# B&R Automation Studio project NAINV104C00R8L515F00 (part 29)

#### Act_Background_Sequence.st - Do Not Change!!!
```iecst
 (** 2019-05-04 **)
ACTION Act_Background_Sequence:

	IF eStatus1 <> Error THEN

		IF p_bOpsRun = FALSE THEN
			p_bSndIncompl	:= TRUE;
		END_IF

		IF tyMsgTypeRcv.bStopTransport = TRUE THEN
			IF tyStopTransport.tyData.eTransferState = HermesTransferStateNotStarted THEN
				p_bSndNotStart	:= TRUE;
			ELSIF tyStopTransport.tyData.eTransferState = HermesTransferStateIncomplete THEN
				p_bSndIncompl	:= TRUE;
			END_IF
		END_IF

		bBlkDS := p_bHermesSwitchtoRvrseTransport;
		//Sequence
		fbSequenceDS.bRstState		:= bRstState;
		fbSequenceDS.bRdySnd		:= p_bRdySnd;
		fbSequenceDS.bBlkDS			:= bBlkDS;
		fbSequenceDS.bSndCompl		:= p_bSndCompl;
		fbSequenceDS.bSndIncompl	:= p_bSndIncompl;
		fbSequenceDS.bSndNotStart	:= p_bSndNotStart;
		fbSequenceDS.bFeatureBoardForecast	:= bFeatureBoardForecast; //Feature BoardForecast
		fbSequenceDS.bOpsRun	        	:= p_bOpsRun; //Machine in AutoMode
		fbSequenceDS.bSendBFId              := bSendBFId; //Send B.F with forecast ID, then block Hermes.eState until Downstream reply a MachineReady(Id) or MachineReady()
		fbSequenceDS.bBFIdSent              := bBFIdSent;
		fbSequenceDS.bSendBFNoID			:= bSendBFNoID;
		fbSequenceDS(bEn := TRUE);
		bUSRdy			:= fbSequenceDS.bUSRdy;
		bDSRdy			:= fbSequenceDS.bDSRdy;
		bTransporting	:= fbSequenceDS.bTransporting;
		bStopTransport	:= fbSequenceDS.bStopTransport;

		bUSGdRdy	:= (tyBoardAvailableSnd.tyAvl.bFailedBoard = FALSE) OR ((tyBoardAvailableSnd.tyAvl.bFailedBoard = TRUE) AND (tyBoardAvailableSnd.tyData.eFailedBoard <> HermesFailedBoard));

		bDSGdRdy	:= (tyMachineReady.tyAvl.bFailedBoard = FALSE) OR ((tyMachineReady.tyAvl.bFailedBoard = TRUE) AND (tyMachineReady.tyData.eFailedBoard <> HermesFailedBoard));

		IF fbSequenceDS.eState >= HermesStateNotAvailableNotReady THEN
			bHandshakeDone	:= TRUE;
		ELSE
			bHandshakeDone	:= FALSE;
		END_IF

		IF EDGEPOS(fbSequenceDS.eState = HermesStateTransporting) THEN
			p_bSndCompl		:= FALSE;
			p_bSndIncompl	:= FALSE;
			p_bSndNotStart	:= FALSE;
		END_IF

		IF fbSequenceDS.eMsgTypeSnd = HermesMsgTypeServiceDescription THEN
			fHermesAddOneMsgSend(ADR(a_eMsgSend) , ADR(udiMsgSendBffr) , HermesMsgTypeServiceDescription);

			tyServiceDescriptionSnd.tyData.sMachineId								    	:= p_sMcId;
			tyServiceDescriptionSnd.tyData.iLaneId											:= p_tyParam.iLaneID;
			tyServiceDescriptionSnd.tyData.sInterfaceId										:= p_sInterfaceId;
			tyServiceDescriptionSnd.tyData.sVersion											:= p_sVersion;
			tyServiceDescriptionSnd.tyData.tySupportedFeatures.bFeatureCheckAliveResponse	:= (p_tyParam.bFeatureCheckAliveResponse) AND (p_tyParam.tRcvAlive <> T#0s) AND (p_tyParam.tSndAlive <> T#0s);
			tyServiceDescriptionSnd.tyData.tySupportedFeatures.bFeatureBoardForecast		:= p_tyParam.bFeatureBoardForecast;
			tyServiceDescriptionSnd.tyData.tySupportedFeatures.bFeatureQueryBoardInfo		:= FALSE;
			tyServiceDescriptionSnd.tyData.tySupportedFeatures.bFeatureSendBoardInfo		:= p_tyParam.bFeatureSendBoardInfo;
			tyServiceDescriptionSnd.tyData.tySupportedFeatures.bFeatureCommand				:= p_tyParam.bFeatureCommand;

			tyServiceDescriptionSnd.tyAvl.bMachineId										:= tyServiceDescriptionSnd.tyData.sMachineId <> '';
			tyServiceDescriptionSnd.tyAvl.bLaneId											:= tyServiceDescriptionSnd.tyData.iLaneId<>0;
			tyServiceDescriptionSnd.tyAvl.bInterfaceId										:= tyServiceDescriptionSnd.tyData.sInterfaceId <> '';
			tyServiceDescriptionSnd.tyAvl.bVersion											:= TRUE;
			tyServiceDescriptionSnd.tyAvl.bSupportedFeatures								:= p_tyParam.bFeatureCheckAliveResponse OR p_tyParam.bFeatureBoardForecast OR p_tyParam.bFeatureSendBoardInfo OR p_tyParam.bFeatureCommand;
			tyServiceDescriptionSnd.tyAvl.tySupportedFeatures.bFeatureCheckAliveResponse	:= (p_tyParam.bFeatureCheckAliveResponse) AND (p_tyParam.tRcvAlive <> T#0s) AND (p_tyParam.tSndAlive <> T#0s);
			tyServiceDescriptionSnd.tyAvl.tySupportedFeatures.bFeatureBoardForecast			:= p_tyParam.bFeatureBoardForecast;
			tyServiceDescriptionSnd.tyAvl.tySupportedFeatures.bFeatureQueryBoardInfo		:= FALSE;
			tyServiceDescriptionSnd.tyAvl.tySupportedFeatures.bFeatureSendBoardInfo			:= p_tyParam.bFeatureSendBoardInfo;
			tyServiceDescriptionSnd.tyAvl.tySupportedFeatures.bFeatureCommand				:= p_tyParam.bFeatureCommand;
		ELSIF fbSequenceDS.eMsgTypeSnd = HermesMsgTypeBoardForecastId THEN //Properties changed
			//need to mantain at one
			fHermesAddOneMsgSend(ADR(a_eMsgSend) , ADR(udiMsgSendBffr) , HermesMsgTypeBoardForecast);
			fHermesGenerateUUID(ADR(tyBoardForecastSnd.tyData.sForecastId) , p_tyDTStructure , pa_usiMacAddr); //Generate ForecastID if there is new Product Changeover
			bBFIdSent := TRUE;

			IF p_bManualInsertData = FALSE THEN //insert board function (from SvyHermes)
				tyBoardForecastSnd.tyData.rTimeUntilAvailable       := p_rMcCycleTm + p_rAWCycleTm;
				tyBoardForecastSnd.tyData.sBoardId 			        := ''; //no need to send BoardId for HermesMsgTypeBoardForecastId.
				tyBoardForecastSnd.tyData.sBoardIdCreatedBy			:= ''; //no need to send BoardIdCreatedBy since no BoardId.
				tyBoardForecastSnd.tyData.eFailedBoard 			    := p_eFailedBoard;
				tyBoardForecastSnd.tyData.sProductTypeId 			:= p_sRecipeNm; //recipe0 name = running recipe name
				tyBoardForecastSnd.tyData.eFlippedBoard 			:= p_eFlippedBoard;
				tyBoardForecastSnd.tyData.sTopBarcode 		    	:= p_sTopBarcode;
				tyBoardForecastSnd.tyData.sBottomBarcode 			:= p_sBottomBarcode;
				tyBoardForecastSnd.tyData.rLength 				    := p_rLength;
				tyBoardForecastSnd.tyData.rWidth 			    	:= DINT_TO_REAL(p_diWidthInUM) / 1000; //recipe 0 width	 = running recipe width
				tyBoardForecastSnd.tyData.rThickness 		    	:= p_rThickness;
				tyBoardForecastSnd.tyData.rConveyorSpeed 			:= p_rConveyorSpeed;
				tyBoardForecastSnd.tyData.rTopClearanceHeight 		:= p_rTopClearanceHeight;
				tyBoardForecastSnd.tyData.rBottomClearanceHeight 	:= p_rBottomClearanceHeight;
				tyBoardForecastSnd.tyData.rWeight 			    	:= p_rWeight;
				tyBoardForecastSnd.tyData.sWorkOrderId 			    := p_sWorkOrderId;
				tyBoardForecastSnd.tyData.sBatchId 			        := p_sBatchId;

				tyBoardForecastSnd.tyAvl.bForecastId 			    := TRUE;
				tyBoardForecastSnd.tyAvl.bTimeUntilAvailable		:= tyBoardForecastSnd.tyData.rTimeUntilAvailable <> 0;
				tyBoardForecastSnd.tyAvl.bBoardId 				    := tyBoardForecastSnd.tyData.sBoardId <> '';
				tyBoardForecastSnd.tyAvl.bBoardIdCreatedBy 		    := TRUE;
				tyBoardForecastSnd.tyAvl.bFailedBoard 			    := TRUE;
				tyBoardForecastSnd.tyAvl.bProductTypeId 			:= tyBoardForecastSnd.tyData.sProductTypeId <> '';
				tyBoardForecastSnd.tyAvl.bFlippedBoard 			    := TRUE;
				tyBoardForecastSnd.tyAvl.bTopBarcode 			    := tyBoardForecastSnd.tyData.sTopBarcode <> '';
				tyBoardForecastSnd.tyAvl.bBottomBarcode 			:= tyBoardForecastSnd.tyData.sBottomBarcode <> '';
				tyBoardForecastSnd.tyAvl.bLength 				    := tyBoardForecastSnd.tyData.rLength <> 0;
				tyBoardForecastSnd.tyAvl.bWidth 				    := tyBoardForecastSnd.tyData.rWidth <> 0 AND (p_bBFWidthEn = TRUE);
				tyBoardForecastSnd.tyAvl.bThickness 			    := tyBoardForecastSnd.tyData.rThickness <> 0 AND (p_bBFSltEn = TRUE);
				tyBoardForecastSnd.tyAvl.bConveyorSpeed 			:= tyBoardForecastSnd.tyData.rConveyorSpeed <> 0;
				tyBoardForecastSnd.tyAvl.bTopClearanceHeight 		:= tyBoardForecastSnd.tyData.rTopClearanceHeight <> 0 AND (p_bBFSltEn = TRUE);
				tyBoardForecastSnd.tyAvl.bBottomClearanceHeight 	:= tyBoardForecastSnd.tyData.rBottomClearanceHeight <> 0 AND (p_bBFSltEn = TRUE);
				tyBoardForecastSnd.tyAvl.bWeight 			    	:= tyBoardForecastSnd.tyData.rWeight <> 0;
				tyBoardForecastSnd.tyAvl.bWorkOrderId 		    	:= tyBoardForecastSnd.tyData.sWorkOrderId <> '';
				tyBoardForecastSnd.tyAvl.bBatchId 		        	:= tyBoardForecastSnd.tyData.sBatchId <> '';
			ELSE //from Rcp
				tyBoardForecastSnd.tyData.rTimeUntilAvailable       := p_rMcCycleTm + p_rAWCycleTm;
				tyBoardForecastSnd.tyData.sBoardId 			        := ''; //no need to send BoardId for HermesMsgTypeBoardForecastId.
				tyBoardForecastSnd.tyData.sBoardIdCreatedBy			:= ''; //no need to send BoardIdCreatedBy since no BoardId.
				tyBoardForecastSnd.tyData.eFailedBoard 			    := p_tySvyHermesSendWorkOrderInfo.tyData.eFailedBoard;
				tyBoardForecastSnd.tyData.sProductTypeId 			:= p_tySvyHermesSendWorkOrderInfo.tyData.sProductTypeId;
				tyBoardForecastSnd.tyData.eFlippedBoard 			:= p_tySvyHermesSendWorkOrderInfo.tyData.eFlippedBoard;
				tyBoardForecastSnd.tyData.sTopBarcode 		    	:= p_tySvyHermesSendWorkOrderInfo.tyData.sTopBarcode;
				tyBoardForecastSnd.tyData.sBottomBarcode 			:= p_tySvyHermesSendWorkOrderInfo.tyData.sBottomBarcode;
				tyBoardForecastSnd.tyData.rLength 				    := p_tySvyHermesSendWorkOrderInfo.tyData.rLength;
				tyBoardForecastSnd.tyData.rWidth 			    	:= DINT_TO_REAL(p_diWidthInUM) / 1000; //recipe 0 width	 = running recipe width
				tyBoardForecastSnd.tyData.rThickness 		    	:= p_tySvyHermesSendWorkOrderInfo.tyData.rThickness;
				tyBoardForecastSnd.tyData.rConveyorSpeed 			:= p_tySvyHermesSendWorkOrderInfo.tyData.rConveyorSpeed;
				tyBoardForecastSnd.tyData.rTopClearanceHeight 		:= p_tySvyHermesSendWorkOrderInfo.tyData.rTopClearanceHeight;
				tyBoardForecastSnd.tyData.rBottomClearanceHeight 	:= p_tySvyHermesSendWorkOrderInfo.tyData.rBottomClearanceHeight;
				tyBoardForecastSnd.tyData.rWeight 			    	:= p_tySvyHermesSendWorkOrderInfo.tyData.rWeight;
				tyBoardForecastSnd.tyData.sWorkOrderId 			    := p_tySvyHermesSendWorkOrderInfo.tyData.sWorkOrderId;
				tyBoardForecastSnd.tyData.sBatchId 			        := p_tySvyHermesSendWorkOrderInfo.tyData.sBatchId;

				tyBoardForecastSnd.tyAvl.bForecastId 			    := TRUE;
				tyBoardForecastSnd.tyAvl.bTimeUntilAvailable		:= tyBoardForecastSnd.tyData.rTimeUntilAvailable <> 0;
				tyBoardForecastSnd.tyAvl.bBoardId 				    := tyBoardForecastSnd.tyData.sBoardId <> '';
				tyBoardForecastSnd.tyAvl.bBoardIdCreatedBy 		    := TRUE;
				tyBoardForecastSnd.tyAvl.bFailedBoard 			    := TRUE;
				tyBoardForecastSnd.tyAvl.bProductTypeId 			:= tyBoardForecastSnd.tyData.sProductTypeId <> '';
				tyBoardForecastSnd.tyAvl.bFlippedBoard 			    := TRUE;
				tyBoardForecastSnd.tyAvl.bTopBarcode 			    := tyBoardForecastSnd.tyData.sTopBarcode <> '';
				tyBoardForecastSnd.tyAvl.bBottomBarcode 			:= tyBoardForecastSnd.tyData.sBottomBarcode <> '';
				tyBoardForecastSnd.tyAvl.bLength 				    := tyBoardForecastSnd.tyData.rLength <> 0;
				tyBoardForecastSnd.tyAvl.bWidth 				    := tyBoardForecastSnd.tyData.rWidth <> 0 AND (p_bBFWidthEn = TRUE);
				tyBoardForecastSnd.tyAvl.bThickness 			    := tyBoardForecastSnd.tyData.rThickness <> 0 AND (p_bBFSltEn = TRUE);
				tyBoardForecastSnd.tyAvl.bConveyorSpeed 			:= tyBoardForecastSnd.tyData.rConveyorSpeed <> 0;
				tyBoardForecastSnd.tyAvl.bTopClearanceHeight 		:= tyBoardForecastSnd.tyData.rTopClearanceHeight <> 0 AND (p_bBFSltEn = TRUE);
				tyBoardForecastSnd.tyAvl.bBottomClearanceHeight 	:= tyBoardForecastSnd.tyData.rBottomClearanceHeight <> 0 AND (p_bBFSltEn = TRUE);
				tyBoardForecastSnd.tyAvl.bWeight 			    	:= tyBoardForecastSnd.tyData.rWeight <> 0;
				tyBoardForecastSnd.tyAvl.bWorkOrderId 		    	:= tyBoardForecastSnd.tyData.sWorkOrderId <> '';
				tyBoardForecastSnd.tyAvl.bBatchId 		        	:= tyBoardForecastSnd.tyData.sBatchId <> '';

			END_IF

		ELSIF fbSequenceDS.eMsgTypeSnd = HermesMsgTypeBoardForecastNoId THEN
			//do not need to count
			fHermesAddOneMsgSend(ADR(a_eMsgSend) , ADR(udiMsgSendBffr) , HermesMsgTypeBoardForecast);
			tyBoardForecastSnd.tyData.sForecastId		        := ''; //Do not need to generate ForecastID to downstream

			IF p_bNewBrdAvlFirstZone AND p_bManualInsertData = FALSE THEN
				fHermesGenerateUUID(ADR(tyBoardForecastSnd.tyData.sBoardId) , p_tyDTStructure , pa_usiMacAddr);
				tyBoardForecastSnd.tyData.sBoardIdCreatedBy         := p_sMcId;
				tyBoardForecastSnd.tyData.eFailedBoard 		    	:= p_eFailedBoard;
				tyBoardForecastSnd.tyData.sProductTypeId 			:= p_sRecipeNm;	 //recipe 0 name = running recipe name
				tyBoardForecastSnd.tyData.eFlippedBoard 			:= p_eFlippedBoard;
				tyBoardForecastSnd.tyData.sTopBarcode 		    	:= p_sTopBarcode;
				tyBoardForecastSnd.tyData.sBottomBarcode 			:= p_sBottomBarcode;
				tyBoardForecastSnd.tyData.rLength 				    := p_rLength;
				tyBoardForecastSnd.tyData.rWidth 			    	:= DINT_TO_REAL(p_diWidthInUM) / 1000;	//recipe 0 width = running recipe width
				tyBoardForecastSnd.tyData.rThickness 		    	:= p_rThickness;
				tyBoardForecastSnd.tyData.rConveyorSpeed 			:= p_rConveyorSpeed;
				tyBoardForecastSnd.tyData.rTopClearanceHeight 		:= p_rTopClearanceHeight;
				tyBoardForecastSnd.tyData.rBottomClearanceHeight 	:= p_rBottomClearanceHeight;
				tyBoardForecastSnd.tyData.rWeight 			    	:= p_rWeight;
				tyBoardForecastSnd.tyData.sWorkOrderId 		    	:= p_sWorkOrderId;
				tyBoardForecastSnd.tyData.sBatchId	    	    	:= p_sBatchId;

				tyBoardForecastSnd.tyAvl.bForecastId 			    := tyBoardForecastSnd.tyData.sForecastId <> '';
				tyBoardForecastSnd.tyAvl.bTimeUntilAvailable		:= tyBoardForecastSnd.tyData.rTimeUntilAvailable <> 0;
				tyBoardForecastSnd.tyAvl.bBoardId 				    := tyBoardForecastSnd.tyData.sBoardId <> '';
				tyBoardForecastSnd.tyAvl.bBoardIdCreatedBy 	    	:= tyBoardForecastSnd.tyData.sBoardIdCreatedBy <> '';
				tyBoardForecastSnd.tyAvl.bFailedBoard 			    := TRUE;
				tyBoardForecastSnd.tyAvl.bProductTypeId 			:= tyBoardForecastSnd.tyData.sProductTypeId <> '';
				tyBoardForecastSnd.tyAvl.bFlippedBoard 		    	:= TRUE;
				tyBoardForecastSnd.tyAvl.bTopBarcode 			    := tyBoardForecastSnd.tyData.sTopBarcode <> '';
				tyBoardForecastSnd.tyAvl.bBottomBarcode 			:= tyBoardForecastSnd.tyData.sBottomBarcode <> '';
				tyBoardForecastSnd.tyAvl.bLength 				    := tyBoardForecastSnd.tyData.rLength <> 0;
				tyBoardForecastSnd.tyAvl.bWidth 				    := tyBoardForecastSnd.tyData.rWidth <> 0 AND (p_bBFWidthEn = TRUE);
				tyBoardForecastSnd.tyAvl.bThickness 			    := tyBoardForecastSnd.tyData.rThickness <> 0 AND (p_bBFSltEn = TRUE);
				tyBoardForecastSnd.tyAvl.bConveyorSpeed 			:= tyBoardForecastSnd.tyData.rConveyorSpeed <> 0;
				tyBoardForecastSnd.tyAvl.bTopClearanceHeight 		:= tyBoardForecastSnd.tyData.rTopClearanceHeight <>0 AND (p_bBFSltEn = TRUE);
				tyBoardForecastSnd.tyAvl.bBottomClearanceHeight 	:= tyBoardForecastSnd.tyData.rBottomClearanceHeight <>0 AND (p_bBFSltEn = TRUE);
				tyBoardForecastSnd.tyAvl.bWeight 			    	:= tyBoardForecastSnd.tyData.rWeight <> 0;
				tyBoardForecastSnd.tyAvl.bWorkOrderId 		    	:= tyBoardForecastSnd.tyData.sWorkOrderId <> '';
				tyBoardForecastSnd.tyAvl.bBatchId 		        	:= tyBoardForecastSnd.tyData.sBatchId <> '';
			ELSIF p_bNewBrdAvlFirstZone AND p_bManualInsertData THEN //insert board data
				fHermesGenerateUUID(ADR(tyBoardForecastSnd.tyData.sBoardId) , p_tyDTStructure , pa_usiMacAddr);
				tyBoardForecastSnd.tyData.sBoardIdCreatedBy         := p_sMcId;
				tyBoardForecastSnd.tyData.eFailedBoard 		    	:= p_tySvyHermesSendWorkOrderInfo.tyData.eFailedBoard;
				tyBoardForecastSnd.tyData.sProductTypeId 			:= p_tySvyHermesSendWorkOrderInfo.tyData.sProductTypeId;
				tyBoardForecastSnd.tyData.eFlippedBoard 			:= p_tySvyHermesSendWorkOrderInfo.tyData.eFlippedBoard;
				tyBoardForecastSnd.tyData.sTopBarcode 		    	:= p_tySvyHermesSendWorkOrderInfo.tyData.sTopBarcode;
				tyBoardForecastSnd.tyData.sBottomBarcode 			:= p_tySvyHermesSendWorkOrderInfo.tyData.sBottomBarcode;
				tyBoardForecastSnd.tyData.rLength 				    := p_tySvyHermesSendWorkOrderInfo.tyData.rLength;
				tyBoardForecastSnd.tyData.rWidth 			    	:= DINT_TO_REAL(p_diWidthInUM) / 1000;	//recipe 0 width = running recipe width
				tyBoardForecastSnd.tyData.rThickness 		    	:= p_tySvyHermesSendWorkOrderInfo.tyData.rThickness;
				tyBoardForecastSnd.tyData.rConveyorSpeed 			:= p_tySvyHermesSendWorkOrderInfo.tyData.rConveyorSpeed;
				tyBoardForecastSnd.tyData.rTopClearanceHeight 		:= p_tySvyHermesSendWorkOrderInfo.tyData.rTopClearanceHeight;
				tyBoardForecastSnd.tyData.rBottomClearanceHeight 	:= p_tySvyHermesSendWorkOrderInfo.tyData.rBottomClearanceHeight;
				tyBoardForecastSnd.tyData.rWeight 			    	:= p_tySvyHermesSendWorkOrderInfo.tyData.rWeight;
				tyBoardForecastSnd.tyData.sWorkOrderId 		    	:= p_tySvyHermesSendWorkOrderInfo.tyData.sWorkOrderId;
				tyBoardForecastSnd.tyData.sBatchId	    	    	:= p_tySvyHermesSendWorkOrderInfo.tyData.sBatchId;

				tyBoardForecastSnd.tyAvl.bForecastId 			    := tyBoardForecastSnd.tyData.sForecastId <> '';
				tyBoardForecastSnd.tyAvl.bTimeUntilAvailable		:= tyBoardForecastSnd.tyData.rTimeUntilAvailable <> 0;
				tyBoardForecastSnd.tyAvl.bBoardId 				    := tyBoardForecastSnd.tyData.sBoardId <> '';
				tyBoardForecastSnd.tyAvl.bBoardIdCreatedBy 	    	:= tyBoardForecastSnd.tyData.sBoardIdCreatedBy <> '';
				tyBoardForecastSnd.tyAvl.bFailedBoard 			    := TRUE;
				tyBoardForecastSnd.tyAvl.bProductTypeId 			:= tyBoardForecastSnd.tyData.sProductTypeId <> '';
				tyBoardForecastSnd.tyAvl.bFlippedBoard 		    	:= TRUE;
				tyBoardForecastSnd.tyAvl.bTopBarcode 			    := tyBoardForecastSnd.tyData.sTopBarcode <> '';
				tyBoardForecastSnd.tyAvl.bBottomBarcode 			:= tyBoardForecastSnd.tyData.sBottomBarcode <> '';
				tyBoardForecastSnd.tyAvl.bLength 				    := tyBoardForecastSnd.tyData.rLength <> 0;
				tyBoardForecastSnd.tyAvl.bWidth 				    := tyBoardForecastSnd.tyData.rWidth <> 0 AND (p_bBFWidthEn = TRUE);
				tyBoardForecastSnd.tyAvl.bThickness 			    := tyBoardForecastSnd.tyData.rThickness <> 0 AND (p_bBFSltEn = TRUE);
				tyBoardForecastSnd.tyAvl.bConveyorSpeed 			:= tyBoardForecastSnd.tyData.rConveyorSpeed <> 0;
				tyBoardForecastSnd.tyAvl.bTopClearanceHeight 		:= tyBoardForecastSnd.tyData.rTopClearanceHeight <>0 AND (p_bBFSltEn = TRUE);
				tyBoardForecastSnd.tyAvl.bBottomClearanceHeight 	:= tyBoardForecastSnd.tyData.rBottomClearanceHeight <>0 AND (p_bBFSltEn = TRUE);
				tyBoardForecastSnd.tyAvl.bWeight 			    	:= tyBoardForecastSnd.tyData.rWeight <> 0;
				tyBoardForecastSnd.tyAvl.bWorkOrderId 		    	:= tyBoardForecastSnd.tyData.sWorkOrderId <> '';
				tyBoardForecastSnd.tyAvl.bBatchId 		        	:= tyBoardForecastSnd.tyData.sBatchId <> '';
			ELSIF p_bNewBrdAvlFirstZone AND bSendBFNoID THEN //Tigger by US hermes to Reverse DS Hermes
				fHermesAddOneMsgSend(ADR(a_eMsgSend) , ADR(udiMsgSendBffr) , HermesMsgTypeBoardForecast);
				IF EDGEPOS(bSndReverseBF) THEN //up pulse trigger with BrdId
					fbParseBrdAvlExternal.p_XMLTable		:= ADR(pa_RevtyXMLTableDataBrdAvl);//last zone B.A
					fbParseBrdAvlExternal.iTotalIdxWrite	:= p_ReviXMLTableDataBrdAvlTtlIdx; //last zone
					fbParseBrdAvlExternal;
					fHermesBrdAvltoBF(ADR(tyBoardForecastSnd),ADR(fbParseBrdAvlExternal.tyBoardAvailable));
				ELSIF EDGENEG(bSndReverseBF) THEN //downpulse , reset
					memset(ADR(tyBoardForecastSnd),0,SIZEOF(tyBoardForecastSnd));
				END_IF
			ELSE   //have brd detail

				//fBrdAvltoBFcast(ADR(),ADR());
				tyBoardForecastSnd.tyData.sBoardId                  := p_tyUSBoardArrivedData.tyData.sBoardId;
				tyBoardForecastSnd.tyData.sBoardIdCreatedBy         := p_tyUSBoardArrivedData.tyData.sBoardIdCreatedBy;
				tyBoardForecastSnd.tyData.eFailedBoard 		    	:= p_tyUSBoardArrivedData.tyData.eFailedBoard;
				tyBoardForecastSnd.tyData.sProductTypeId 			:= p_tyUSBoardArrivedData.tyData.sProductTypeId;
				tyBoardForecastSnd.tyData.eFlippedBoard 			:= p_tyUSBoardArrivedData.tyData.eFlippedBoard;
				tyBoardForecastSnd.tyData.sTopBarcode 		    	:= p_tyUSBoardArrivedData.tyData.sTopBarcode;
				tyBoardForecastSnd.tyData.sBottomBarcode 			:= p_tyUSBoardArrivedData.tyData.sBottomBarcode;
				tyBoardForecastSnd.tyData.rLength 				    := p_tyUSBoardArrivedData.tyData.rLength;
				tyBoardForecastSnd.tyData.rWidth 			    	:= p_tyUSBoardArrivedData.tyData.rWidth;
				tyBoardForecastSnd.tyData.rThickness 		    	:= p_tyUSBoardArrivedData.tyData.rThickness;
				tyBoardForecastSnd.tyData.rConveyorSpeed 			:= p_tyUSBoardArrivedData.tyData.rConveyorSpeed;
				tyBoardForecastSnd.tyData.rTopClearanceHeight 		:= p_tyUSBoardArrivedData.tyData.rTopClearanceHeight;
				tyBoardForecastSnd.tyData.rBottomClearanceHeight 	:= p_tyUSBoardArrivedData.tyData.rBottomClearanceHeight;
				tyBoardForecastSnd.tyData.rWeight 			    	:= p_tyUSBoardArrivedData.tyData.rWeight;
				tyBoardForecastSnd.tyData.sWorkOrderId 		    	:= p_tyUSBoardArrivedData.tyData.sWorkOrderId;
				tyBoardForecastSnd.tyData.sBatchId 		        	:= p_tyUSBoardArrivedData.tyData.sBatchId;

				tyBoardForecastSnd.tyAvl.bForecastId 			    := tyBoardForecastSnd.tyData.sForecastId <> '';
				tyBoardForecastSnd.tyAvl.bTimeUntilAvailable		:= tyBoardForecastSnd.tyData.rTimeUntilAvailable <> 0;
				tyBoardForecastSnd.tyAvl.bBoardId 				    := tyBoardForecastSnd.tyData.sBoardId <> '';
				tyBoardForecastSnd.tyAvl.bBoardIdCreatedBy 	    	:= tyBoardForecastSnd.tyData.sBoardIdCreatedBy <> '';
				tyBoardForecastSnd.tyAvl.bFailedBoard 			    := TRUE;
				tyBoardForecastSnd.tyAvl.bProductTypeId 			:= tyBoardForecastSnd.tyData.sProductTypeId <> '';
				tyBoardForecastSnd.tyAvl.bFlippedBoard 		    	:= TRUE;
				tyBoardForecastSnd.tyAvl.bTopBarcode 			    := tyBoardForecastSnd.tyData.sTopBarcode <> '';
				tyBoardForecastSnd.tyAvl.bBottomBarcode 			:= tyBoardForecastSnd.tyData.sBottomBarcode <> '';
				tyBoardForecastSnd.tyAvl.bLength 				    := tyBoardForecastSnd.tyData.rLength <> 0;
				tyBoardForecastSnd.tyAvl.bWidth 				    := tyBoardForecastSnd.tyData.rWidth <> 0;
				tyBoardForecastSnd.tyAvl.bThickness 			    := tyBoardForecastSnd.tyData.rThickness <> 0;
				tyBoardForecastSnd.tyAvl.bConveyorSpeed 			:= tyBoardForecastSnd.tyData.rConveyorSpeed <> 0;
				tyBoardForecastSnd.tyAvl.bTopClearanceHeight 		:= tyBoardForecastSnd.tyData.rTopClearanceHeight <> 0;
				tyBoardForecastSnd.tyAvl.bBottomClearanceHeight 	:= tyBoardForecastSnd.tyData.rBottomClearanceHeight <> 0;
				tyBoardForecastSnd.tyAvl.bWeight 			    	:= tyBoardForecastSnd.tyData.rWeight <> 0;
				tyBoardForecastSnd.tyAvl.bWorkOrderId 		    	:= tyBoardForecastSnd.tyData.sWorkOrderId <> '';
				tyBoardForecastSnd.tyAvl.bBatchId 		        	:= tyBoardForecastSnd.tyData.sBatchId <> '';

			END_IF
		ELSIF fbSequenceDS.eMsgTypeSnd = HermesMsgTypeBoardAvailable THEN
			fHermesAddOneMsgSend(ADR(a_eMsgSend) , ADR(udiMsgSendBffr) , HermesMsgTypeBoardAvailable);

			tyBoardAvailableSnd.tyData.iRoute	:= iRoute;
			tyBoardAvailableSnd.tyData.iAction	:= iAction;

			tyBoardAvailableSnd.tyAvl.bRoute := tyBoardAvailableSnd.tyData.iRoute <> 0;
			tyBoardAvailableSnd.tyAvl.bAction:= tyBoardAvailableSnd.tyData.iAction <> 0 ;

			IF p_bNewBrdAvlLastZone = TRUE AND p_bRcvBoardInfo = FALSE THEN //Generate New B.A for Unknown PCB
				IF bFeatureBoardForecast AND bBFIdSent THEN
					tyBoardAvailableSnd.tyData.sBoardId :=	 tyBoardForecastSnd.tyData.sBoardId;
				ELSE
					fHermesGenerateUUID(ADR(tyBoardAvailableSnd.tyData.sBoardId) , p_tyDTStructure , pa_usiMacAddr);
				END_IF

				tyBoardAvailableSnd.tyData.sBoardIdCreatedBy        := p_sMcId; //Generate by our Machine
				tyBoardAvailableSnd.tyData.eFailedBoard				:= p_eFailedBoard;
				tyBoardAvailableSnd.tyData.sProductTypeId			:= p_sRecipeNm;
				tyBoardAvailableSnd.tyData.eFlippedBoard			:= p_eFlippedBoard;
				tyBoardAvailableSnd.tyData.sTopBarcode				:= p_sTopBarcode;
				tyBoardAvailableSnd.tyData.sBottomBarcode			:= p_sBottomBarcode;
				tyBoardAvailableSnd.tyData.rLength					:= p_rLength;
				tyBoardAvailableSnd.tyData.rWidth					:= DINT_TO_REAL(p_diWidthInUM) / 1000;
				tyBoardAvailableSnd.tyData.rThickness				:= p_rThickness;
				tyBoardAvailableSnd.tyData.rConveyorSpeed			:= p_rConveyorSpeed;
				tyBoardAvailableSnd.tyData.rTopClearanceHeight		:= p_rTopClearanceHeight;
				tyBoardAvailableSnd.tyData.rBottomClearanceHeight	:= p_rBottomClearanceHeight;
				tyBoardAvailableSnd.tyData.rWeight					:= p_rWeight;
				tyBoardAvailableSnd.tyData.sWorkOrderId			    := p_sWorkOrderId;
				tyBoardAvailableSnd.tyData.sBatchId			        := p_sBatchId;

				tyBoardAvailableSnd.tyAvl.bBoardId					:= tyBoardAvailableSnd.tyData.sBoardId<>'';
				tyBoardAvailableSnd.tyAvl.bBoardIdCreatedBy			:= tyBoardAvailableSnd.tyData.sBoardIdCreatedBy <> '';
				tyBoardAvailableSnd.tyAvl.bFailedBoard				:= TRUE;
				tyBoardAvailableSnd.tyAvl.bProductTypeId			:= tyBoardAvailableSnd.tyData.sProductTypeId <> '';
				tyBoardAvailableSnd.tyAvl.bFlippedBoard				:= TRUE;
				tyBoardAvailableSnd.tyAvl.bTopBarcode				:= tyBoardAvailableSnd.tyData.sTopBarcode <> '';
				tyBoardAvailableSnd.tyAvl.bBottomBarcode			:= tyBoardAvailableSnd.tyData.sBottomBarcode <> '';
				tyBoardAvailableSnd.tyAvl.bLength					:= tyBoardAvailableSnd.tyData.rLength <> 0;
				tyBoardAvailableSnd.tyAvl.bWidth					:= (tyBoardAvailableSnd.tyData.rWidth <> 0) AND (p_bBAWidthEn = TRUE);
				tyBoardAvailableSnd.tyAvl.bThickness				:= (tyBoardAvailableSnd.tyData.rThickness <> 0) AND (p_bBASltEn = TRUE);
				tyBoardAvailableSnd.tyAvl.bConveyorSpeed			:= tyBoardAvailableSnd.tyData.rConveyorSpeed <> 0;
				tyBoardAvailableSnd.tyAvl.bTopClearanceHeight		:= (tyBoardAvailableSnd.tyData.rTopClearanceHeight <> 0) AND (p_bBASltEn = TRUE);
				tyBoardAvailableSnd.tyAvl.bBottomClearanceHeight	:= (tyBoardAvailableSnd.tyData.rBottomClearanceHeight <> 0) AND (p_bBASltEn = TRUE);
				tyBoardAvailableSnd.tyAvl.bWeight					:= tyBoardAvailableSnd.tyData.rWeight <> 0;
				tyBoardAvailableSnd.tyAvl.bWorkOrderId				:= tyBoardAvailableSnd.tyData.sWorkOrderId <> '';
				tyBoardAvailableSnd.tyAvl.bBatchId			    	:= tyBoardAvailableSnd.tyData.sBatchId <> '';

			ELSIF p_bNewBrdAvlLastZone = TRUE AND p_bRcvBoardInfo = TRUE THEN //Take BoardInfo From "SendBoardInfo", for Manual Insert PCB

				tyBoardAvailableSnd.tyData.sBoardId                 := p_tyBoardInfoData.tyData.sBoardId;
				tyBoardAvailableSnd.tyData.sBoardIdCreatedBy        := p_tyBoardInfoData.tyData.sBoardIdCreatedBy;
				tyBoardAvailableSnd.tyData.eFailedBoard				:= p_tyBoardInfoData.tyData.eFailedBoard;
				tyBoardAvailableSnd.tyData.sProductTypeId			:= p_tyBoardInfoData.tyData.sProductTypeId;
				tyBoardAvailableSnd.tyData.eFlippedBoard			:= p_tyBoardInfoData.tyData.eFlippedBoard;
				tyBoardAvailableSnd.tyData.sTopBarcode				:= p_tyBoardInfoData.tyData.sTopBarcode;
				tyBoardAvailableSnd.tyData.sBottomBarcode			:= p_tyBoardInfoData.tyData.sBottomBarcode;
				tyBoardAvailableSnd.tyData.rLength					:= p_tyBoardInfoData.tyData.rLength;
				tyBoardAvailableSnd.tyData.rWidth					:= p_tyBoardInfoData.tyData.rWidth;
				tyBoardAvailableSnd.tyData.rThickness				:= p_tyBoardInfoData.tyData.rThickness;
				tyBoardAvailableSnd.tyData.rConveyorSpeed			:= p_rConveyorSpeed; //dont have
				tyBoardAvailableSnd.tyData.rTopClearanceHeight		:= p_tyBoardInfoData.tyData.rTopClearanceHeight;
				tyBoardAvailableSnd.tyData.rBottomClearanceHeight	:= p_tyBoardInfoData.tyData.rBottomClearanceHeight;
				tyBoardAvailableSnd.tyData.rWeight					:= p_tyBoardInfoData.tyData.rWeight;
				tyBoardAvailableSnd.tyData.sWorkOrderId			    := p_tyBoardInfoData.tyData.sWorkOrderId;
				tyBoardAvailableSnd.tyData.sBatchId		            := p_tyBoardInfoData.tyData.sBatchId;

				tyBoardAvailableSnd.tyAvl.bBoardId					:= tyBoardAvailableSnd.tyData.sBoardId <> '';
				tyBoardAvailableSnd.tyAvl.bBoardIdCreatedBy			:= tyBoardAvailableSnd.tyData.sBoardIdCreatedBy <> '';
				tyBoardAvailableSnd.tyAvl.bFailedBoard				:= TRUE;
				tyBoardAvailableSnd.tyAvl.bProductTypeId			:= tyBoardAvailableSnd.tyData.sProductTypeId <> '';
				tyBoardAvailableSnd.tyAvl.bFlippedBoard				:= TRUE;
				tyBoardAvailableSnd.tyAvl.bTopBarcode				:= tyBoardAvailableSnd.tyData.sTopBarcode <> '';
				tyBoardAvailableSnd.tyAvl.bBottomBarcode			:= tyBoardAvailableSnd.tyData.sBottomBarcode <> '';
				tyBoardAvailableSnd.tyAvl.bLength					:= tyBoardAvailableSnd.tyData.rLength <> 0;
				tyBoardAvailableSnd.tyAvl.bWidth					:= (tyBoardAvailableSnd.tyData.rWidth <> 0);
				tyBoardAvailableSnd.tyAvl.bThickness				:= (tyBoardAvailableSnd.tyData.rThickness <> 0);
				tyBoardAvailableSnd.tyAvl.bConveyorSpeed			:= tyBoardAvailableSnd.tyData.rConveyorSpeed <> 0;
				tyBoardAvailableSnd.tyAvl.bTopClearanceHeight		:= (tyBoardAvailableSnd.tyData.rTopClearanceHeight <> 0);
				tyBoardAvailableSnd.tyAvl.bBottomClearanceHeight	:= (tyBoardAvailableSnd.tyData.rBottomClearanceHeight <> 0);
				tyBoardAvailableSnd.tyAvl.bWeight					:= tyBoardAvailableSnd.tyData.rWeight <> 0;
				tyBoardAvailableSnd.tyAvl.bWorkOrderId				:= tyBoardAvailableSnd.tyData.sWorkOrderId <> '';
				tyBoardAvailableSnd.tyAvl.bBatchId			    	:= tyBoardAvailableSnd.tyData.sBatchId <> '';

			ELSE //Take from PCB_In Board Data

				fbParseBrdAvlExternal.p_XMLTable		:= ADR(pa_tyXMLTableDataBrdAvl); //last zone B.A
				fbParseBrdAvlExternal.iTotalIdxWrite	:= p_iXMLTableDataBrdAvlTtlIdx; //last zone
				fbParseBrdAvlExternal;
				tyBoardAvailableSnd	:= fbParseBrdAvlExternal.tyBoardAvailable;
			END_IF

		ELSIF fbSequenceDS.eMsgTypeSnd = HermesMsgTypeRevokeBoardAvl THEN
			fHermesAddOneMsgSend(ADR(a_eMsgSend) , ADR(udiMsgSendBffr) , HermesMsgTypeRevokeBoardAvl);

		ELSIF fbSequenceDS.eMsgTypeSnd = HermesMsgTypeTransportFinished THEN
			fHermesAddOneMsgSend(ADR(a_eMsgSend) , ADR(udiMsgSendBffr) , HermesMsgTypeTransportFinished);

			IF p_bSndCompl = TRUE THEN
				tyTransportFinished.tyData.eTransferState	:= HermesTransferStateComplete;
			ELSIF p_bSndIncompl = TRUE THEN
				tyTransportFinished.tyData.eTransferState	:= HermesTransferStateIncomplete;
			ELSE
				tyTransportFinished.tyData.eTransferState	:= HermesTransferStateNotStarted;
			END_IF
			tyTransportFinished.tyData.sBoardId				:= tyStartTransport.tyData.sBoardId;

			tyTransportFinished.tyAvl.bTransferState		:= TRUE;
			tyTransportFinished.tyAvl.bBoardId				:= TRUE;

		END_IF

	END_IF

END_ACTION
```

#### Act_Background_ChkAliveSendPing.st - Do Not Change!!!
```iecst
(** 2021-08-01 **)
ACTION Act_Background_ChkAliveSendPing:

	IF eStatus1 <> Error THEN

		//Check Alive Send Ping
		fbCheckAliveSendPing.bDataRcv		:= tyMsgTypeRcv.bCheckAlivePong;
		fbCheckAliveSendPing.tyDataRcv		:= tyCheckAlivePongRcv;
		fbCheckAliveSendPing.tyDTStructure	:= p_tyDTStructure;
		fbCheckAliveSendPing.tSendTm		:= p_tyParam.tSndAlive;
		fbCheckAliveSendPing.tRcvTimeOut	:= p_tyParam.tRcvAlive;
		fbCheckAliveSendPing(bEn := TRUE);

		IF fbCheckAliveSendPing.udiStatus > 0 AND fbCheckAliveSendPing.udiStatus < 65534 THEN
			eStatus1	:= Error;

			IF fbCheckAliveSendPing.udiStatus = 2768 THEN
				udiStatus1	:= 10133;	//Waiting Check Alive Time Out
			ELSIF fbCheckAliveSendPing.udiStatus = 2769 THEN
				udiStatus1	:= 10134;	//Check Alive Id Mismatch
			ELSE
				udiStatus1	:= fbCheckAliveSendPing.udiStatus;
			END_IF

			fHermesAddOneMsgSend(ADR(a_eMsgSend) , ADR(udiMsgSendBffr) , HermesMsgTypeNotification);

			tyNotificationSnd.tyAvl.bSeverity			:= TRUE;
			tyNotificationSnd.tyAvl.bNotificationCode	:= TRUE;
			tyNotificationSnd.tyAvl.bDescription		:= TRUE;
			tyNotificationSnd.tyData.eSeverity			:= HermesSeverityFatalError;
			tyNotificationSnd.tyData.iNotificationCode	:= UDINT_TO_INT(udiStatus1);
			tyNotificationSnd.tyData.sDescription		:= a_tyAlmText[udiStatus1].sAlmText;

		ELSE
			IF EDGEPOS(fbCheckAliveSendPing.bDataSend) THEN
				fHermesAddOneMsgSend(ADR(a_eMsgSend) , ADR(udiMsgSendBffr) , HermesMsgTypeCheckAlivePing);
				tyCheckAlivePingSnd	:= fbCheckAliveSendPing.tyDataSend;
			END_IF

		END_IF

		tyMsgTypeRcv.bCheckAlivePong	:= FALSE;	//Reset Check Alive Pong

	END_IF

END_ACTION
```

#### Act_Background_ChkAliveRcvPing.st - Do Not Change!!!
```iecst
(** 2021-08-01 **)
ACTION Act_Background_ChkAliveRcvPing:

	IF eStatus1 <> Error THEN

		//Check Alive Receive Ping
		fbCheckAliveRcvPing.bDataRcv	:= tyMsgTypeRcv.bCheckAlivePing;
		fbCheckAliveRcvPing.tyDataRcv	:= tyCheckAlivePingRcv;
		fbCheckAliveRcvPing(bEn := TRUE);

		IF fbCheckAliveRcvPing.udiStatus > 0 AND fbCheckAliveRcvPing.udiStatus < 65534 THEN
			eStatus1	:= Error;
			udiStatus1	:= fbCheckAliveRcvPing.udiStatus;

		ELSE
			IF EDGEPOS(fbCheckAliveRcvPing.bDataSend) THEN
				fHermesAddOneMsgSend(ADR(a_eMsgSend) , ADR(udiMsgSendBffr) , HermesMsgTypeCheckAlivePong);
				tyCheckAlivePongSnd	:= fbCheckAliveRcvPing.tyDataSend;
			END_IF

		END_IF

		tyMsgTypeRcv.bCheckAlivePing	:= FALSE;	//Reset Check Alive Ping

	END_IF

END_ACTION
```

#### Act_Background_ProcessData.st - Do Not Change!!!
```iecst
(** 2023-08-01 **)
ACTION Act_Background_ProcessData:

	//update from event to trigger message externally
	IF EDGEPOS(eStatus = Done AND eStat = HermesActReadRetain) AND usiBAIndex = 0  THEN //find empty index
		FOR usiBAIndex := 0  TO SIZEOF(a_tyBoardDepartedInfo)/SIZEOF(a_tyBoardDepartedInfo[0]) -1  DO
			IF memcmp(ADR(a_tyBoardDepartedInfo[usiBAIndex].tyData.sBoardId),ADR(''),1) = 0 THEN
				EXIT; //search for index
			END_IF
		END_FOR
		usiPrevBAIndex := usiBAIndex;
	END_IF

	//board departed
	bTransportFinishedSnd := EDGEPOS (fbSequenceDS.eMsgTypeSnd = HermesMsgTypeTransportFinished);

	IF bTransportFinishedSnd THEN
		IF usiBAIndex >= 50 THEN
			usiBAIndex := 0;
		END_IF
		memset(ADR(a_tyBoardDepartedInfo[usiBAIndex]),0,SIZEOF(a_tyBoardDepartedInfo[usiBAIndex]));
		memcpy(ADR(a_tyBoardDepartedInfo[usiBAIndex]),ADR(tyBoardAvailableSnd),SIZEOF(tyBoardAvailableSnd));
		usiBAIndex := usiBAIndex +1;
	END_IF

	IF eStatus = Done AND eStat = HermesActWriteRetain THEN
		eAct			:= HermesActIdle;
		usiPrevBAIndex 	:= usiBAIndex;
	ELSIF eStatus = Idle AND eStat = HermesActIdle  AND  usiPrevBAIndex <> usiBAIndex THEN
		a_tyBoardDepartedInfoWr := a_tyBoardDepartedInfo;
		eAct 					 := HermesActWriteRetain;
	END_IF

END_ACTION
```

#### Act_Background_TCPCloseClnt.st - Do Not Change!!!
```iecst
(** 2019-06-10 **)
ACTION Act_Background_TCPCloseClnt:

	//Close Server Connection
	IF p_bInternalUse = FALSE THEN
		fbCloseClnt.udiTCPIdent	:= udiClntIdent;
		fbCloseClnt(bEn := TRUE);

		IF fbCloseClnt.udiStatus = 0 THEN
			udiClntIdent	:= 0;
			fbCloseClnt(bEn := FALSE);

		ELSIF fbCloseClnt.udiStatus < 65534 THEN
			udiClntIdent	:= 0;
			eStatus1		:= Error;

			IF fbCloseClnt.udiStatus = 2300 THEN
				udiStatus1	:= 10154;	//Invalid Ident While Closing TCP
			ELSIF fbCloseClnt.udiStatus = 2310 THEN
				udiStatus1	:= 10155;	//Closing TCP Error
			ELSE
				udiStatus1	:= fbCloseClnt.udiStatus;
			END_IF

		END_IF

	ELSE
		udiClntIdent	:= 0;

	END_IF

END_ACTION
```

#### Act_Background_Stop.st - Do Not Change!!!
```iecst
(** 2021-08-01 **)
ACTION Act_Background_Stop:

	IF EDGEPOS(bStop) THEN

		fHermesAddOneMsgSend(ADR(a_eMsgSend) , ADR(udiMsgSendBffr) , HermesMsgTypeNotification);

		tyNotificationSnd.tyAvl.bSeverity			:= TRUE;
		tyNotificationSnd.tyAvl.bNotificationCode	:= TRUE;
		tyNotificationSnd.tyAvl.bDescription		:= TRUE;
		tyNotificationSnd.tyData.eSeverity			:= HermesSeverityInfo;
		tyNotificationSnd.tyData.iNotificationCode	:= 5;
		tyNotificationSnd.tyData.sDescription		:= 'Machine Shutdown';

	END_IF

	IF bStop = TRUE THEN

		IF a_eMsgSend[0] = HermesMsgTypeNA THEN

			bRstConnection	:= TRUE;

			IF udiSvrIdent = 0 THEN

				bRun	:= FALSE;

			END_IF

		END_IF

	END_IF

END_ACTION
```

#### Act_Main_Disable.st - Do Not Change!!!
```iecst
(** 2021-08-01 **)
ACTION Act_Main_Disable:

	bConnected		:= FALSE;
	bHandshakeDone	:= FALSE;
	bUSRdy			:= FALSE;
	bDSRdy			:= FALSE;
	bTransporting	:= FALSE;
	bStopTransport	:= FALSE;

END_ACTION
```

#### Act_Alarm2.st - Do Not Change!!!
```iecst
(** 2021-08-01 **)
ACTION Act_Alarm2: //IllegalMsg Check, ChkParamRcv, CmpParamRcv, SequenceTO, B.A Check, B.F Check, bStopTransport

	//Error
	IF EDGEPOS(eStatus2 = Error) THEN

		tyAlmData2.sProgNm		:= p_sProgNm;
		tyAlmData2.udiCode		:= udiStatus2;
		tyAlmData2.eSeverity	:= AlmSeverityError;
		tyAlmData2.udiRunTime	:= tyAlmData2.udiRunTime + 1;
		tyAlmData2.bAlm			:= TRUE;
		tyAlmData2.udiModuleNum := udiModuleNum;
		g_sDSHermesProgNm		:= p_sProgNm;

		//Get Error Message
		IF tyAlmData2.udiCode < 10000 OR tyAlmData2.udiCode > 10199 THEN
			tyAlmData2.sAlmMsg	:= 'Unknown';
			tyAlmData2.sRcyMsg	:= 'Unknown';
		ELSE
			tyAlmData2.sAlmMsg	:= a_tyAlmText[tyAlmData2.udiCode].sAlmText;
			tyAlmData2.sRcyMsg	:= a_tyAlmText[tyAlmData2.udiCode].sRcyText;
		END_IF

		sStatTxt	:= tyAlmData2.sAlmMsg;

	ELSIF bRstErr AND (tyAlmData2.udiCode <> 0) THEN

		tyAlmData2.udiCode		:= 0;
		tyAlmData2.eSeverity	:= AlmSeverityNA;
		tyAlmData2.sAlmMsg		:= '';
		tyAlmData2.sRcyMsg		:= '';
		tyAlmData2.bAlm			:= FALSE;
		sStatTxt	:= a_sStatText[eStat];

	END_IF

END_ACTION
```

#### Act_Alarm3.st - Do Not Change!!!
```iecst
(** 2021-08-01 **)
ACTION Act_Alarm3: //fbFileAppend1 Error

	//Error
	IF EDGEPOS(eStatus3 = Error) THEN

		tyAlmData3.sProgNm		:= p_sProgNm;
		tyAlmData3.udiCode		:= udiStatus3;
		tyAlmData3.eSeverity	:= AlmSeverityError;
		tyAlmData3.udiRunTime	:= tyAlmData3.udiRunTime + 1;
		tyAlmData3.bAlm			:= TRUE;
		tyAlmData3.udiModuleNum  := udiModuleNum;
		g_sDSHermesProgNm		:= p_sProgNm;

		//Get Error Message
		IF tyAlmData3.udiCode < 10000 OR tyAlmData3.udiCode > 10199 THEN
			tyAlmData3.sAlmMsg	:= 'Unknown';
			tyAlmData3.sRcyMsg	:= 'Unknown';
		ELSE
			tyAlmData3.sAlmMsg	:= a_tyAlmText[tyAlmData3.udiCode].sAlmText;
			tyAlmData3.sRcyMsg	:= a_tyAlmText[tyAlmData3.udiCode].sRcyText;
		END_IF

		sStatTxt	:= tyAlmData3.sAlmMsg;

	ELSIF bRstErr AND (tyAlmData3.udiCode <> 0) THEN

		tyAlmData3.udiCode		:= 0;
		tyAlmData3.eSeverity	:= AlmSeverityNA;
		tyAlmData3.sAlmMsg		:= '';
		tyAlmData3.sRcyMsg		:= '';
		tyAlmData3.bAlm			:= FALSE;
		sStatTxt	:= a_sStatText[eStat];

	END_IF

END_ACTION
```

#### Act_Alarm4.st - Do Not Change!!!
```iecst
(** 2021-08-01 **)
ACTION Act_Alarm4: //Not Connected Warning

	//Warning
	IF ((bConnected = FALSE) AND (p_eLinkMcParamDSCommMod= McSetCommModHermes)) THEN

		tyAlmData4.sProgNm		:= p_sProgNm;
		tyAlmData4.udiCode		:= udiStatus4;
		tyAlmData4.eSeverity	:= AlmSeverityWarning;
		tyAlmData4.udiRunTime	:= tyAlmData4.udiRunTime + 1;
		tyAlmData4.bWarning			:= TRUE;
		tyAlmData4.udiModuleNum := udiModuleNum;
		g_sDSHermesProgNm		:= p_sProgNm;

		//Get Warning Message
		IF tyAlmData4.udiCode < 10000 OR tyAlmData4.udiCode > 10199 THEN
			tyAlmData4.sAlmMsg	:= 'Unknown';
			tyAlmData4.sRcyMsg	:= 'Unknown';
		ELSE
			tyAlmData4.sAlmMsg	:= a_tyAlmText[tyAlmData4.udiCode].sAlmText;
			tyAlmData4.sRcyMsg	:= a_tyAlmText[tyAlmData4.udiCode].sRcyText;
		END_IF

		sStatTxt	:= tyAlmData4.sAlmMsg;

	ELSIF (bConnected AND (tyAlmData4.udiCode <> 0)) OR (p_eLinkMcParamDSCommMod= McSetCommModSMEMA) THEN

		tyAlmData4.udiCode		:= 0;
		tyAlmData4.eSeverity	:= AlmSeverityNA;
		tyAlmData4.sAlmMsg		:= '';
		tyAlmData4.sRcyMsg		:= '';
		//tyUIAlmData.bWarning[3363] := FALSE;		// (05042023)Debug Alarm Test
		tyAlmData4.bWarning		:= FALSE;
		sStatTxt	:= a_sStatText[eStat];

	END_IF

END_ACTION
```

#### InputRef.var - Do Not Change!!!
```iecst
(*2019-06-10*)
(**)
(*General*)
VAR
	p_eAct : REFERENCE TO eHermesAction;
	p_udiRstErr : REFERENCE TO UDINT;
	p_bPrep : REFERENCE TO BOOL;
	p_bEn : REFERENCE TO BOOL;
	p_bDis : REFERENCE TO BOOL;
END_VAR
(**)
(*Configuration*)
VAR
	p_tyParam : REFERENCE TO tyHermesDSParam;
	p_sIPAddr : REFERENCE TO STRING[15];
	pa_usiMacAddr : REFERENCE TO ARRAY[0..5] OF USINT;
	p_tyDTStructure : REFERENCE TO DTStructure;
	p_dtCurrDT : REFERENCE TO DATE_AND_TIME;
	p_sMcId : REFERENCE TO STRING[80];
END_VAR
(**)
(*Input*)
VAR
	p_bRdySnd : REFERENCE TO BOOL;
	p_bSndCompl : REFERENCE TO BOOL;
	p_bSndIncompl : REFERENCE TO BOOL;
	p_bSndNotStart : REFERENCE TO BOOL;
	p_bBAWidthEn : REFERENCE TO BOOL; (*Board Available Check Width*)
	p_bBASltEn : REFERENCE TO BOOL; (*Board Available Check Slot*)
	p_bBFWidthEn : REFERENCE TO BOOL; (*Board Forecast Check Width*)
	p_bBFSltEn : REFERENCE TO BOOL; (*Board Forecast Check Slot*)
	p_sRecipeNm : REFERENCE TO STRING[254];
	p_sRecipeZone1Nm : REFERENCE TO STRING[254];
	p_sForecastId : REFERENCE TO STRING[80];
	p_sBoardId : REFERENCE TO STRING[36];
	p_sInterfaceId : REFERENCE TO STRING[80];
	p_sVersion : REFERENCE TO STRING[7];
	p_eFailedBoard : REFERENCE TO eHermesFailedBoard;
	p_eFlippedBoard : REFERENCE TO eHermesFlippedBoard;
	p_sTopBarcode : REFERENCE TO STRING[254];
	p_sBottomBarcode : REFERENCE TO STRING[254];
	p_rLength : REFERENCE TO REAL;
	p_rThickness : REFERENCE TO REAL;
	p_rConveyorSpeed : REFERENCE TO REAL;
	p_rTopClearanceHeight : REFERENCE TO REAL;
	p_rBottomClearanceHeight : REFERENCE TO REAL;
	p_rWeight : REFERENCE TO REAL;
	p_sWorkOrderId : REFERENCE TO STRING[80];
	p_sBatchId : REFERENCE TO STRING[80];
	p_diWidthInUM : REFERENCE TO DINT;
	p_diWidthZone1InUM : REFERENCE TO DINT;
	p_diMinSltValue : REFERENCE TO DINT;
	p_diMaxSltValue : REFERENCE TO DINT;
	p_diPitch : REFERENCE TO DINT;
	p_diTtlSlt : REFERENCE TO DINT;
	p_diSltToSltInUM : REFERENCE TO DINT;
	p_udiSndBffrSize : REFERENCE TO UDINT;
	p_udiRcvBffrSize : REFERENCE TO UDINT;
	p_udiAliveIdleTimeInSec : REFERENCE TO UDINT;
	p_tConnTimeOut : REFERENCE TO TIME;
	p_diTransferInTO : REFERENCE TO DINT;
	pa_tyXMLTableDataBrdAvl1stZ : REFERENCE TO ARRAY[0..200] OF tyXMLTableDat;
	p_iXMLTableDataBrdAvlTtlIdx1stZ : REFERENCE TO INT;
	pa_tyXMLTableDataBrdAvl : REFERENCE TO ARRAY[0..200] OF tyXMLTableDat;
	p_iXMLTableDataBrdAvlTtlIdx : REFERENCE TO INT;
	p_bNewBrdAvlFirstZone : REFERENCE TO BOOL;
	p_bNewBrdAvlLastZone : REFERENCE TO BOOL;
	p_bOpsRun : REFERENCE TO BOOL;
	p_bInterruptSen : REFERENCE TO BOOL;
	p_udiFileKeepDay : REFERENCE TO UDINT;
	p_udiRetainDataAddr : REFERENCE TO UDINT;
	p_udiRetainDataLen : REFERENCE TO UDINT;
	p_sRetainFileName : REFERENCE TO STRING[80];
	p_sProgNm : REFERENCE TO STRING[15];
	p_bNtSettingsLoadDone : REFERENCE TO BOOL;
	p_sRmtMcId : REFERENCE TO STRING[80];
	p_bRmtPrep : REFERENCE TO BOOL;
	p_bRmtEn : REFERENCE TO BOOL;
	p_bUSHermesStopTransport : REFERENCE TO BOOL;
	p_bInternalUse : REFERENCE TO BOOL;
	p_sInternalRcv : REFERENCE TO STRING[65535];
	p_tyUSBoardArrivedData : REFERENCE TO tyHermesBoardAvailable;
	p_bRcvBoardInfo : REFERENCE TO BOOL;
	p_tyBoardInfoData : REFERENCE TO tyHermesSendBoardInfo;
	p_tyUSHermestyBoardAvailable : REFERENCE TO tyHermesBoardAvailable;
	p_bNtParamProjInvertOncePrep : REFERENCE TO BOOL;
	p_bNtParamProjInvertTwicePrep : REFERENCE TO BOOL;
	p_bReverseDSSendBFId : REFERENCE TO BOOL;
	p_rMcCycleTm : REFERENCE TO REAL;
	p_rAWCycleTm : REFERENCE TO REAL;
	p_bConvInitDone : REFERENCE TO BOOL;
END_VAR
(*Reverse Hermes *)
VAR
	p_bManualRmvRoute : REFERENCE TO BOOL;
	p_bReturnRoute : REFERENCE TO BOOL;
	p_bNomRouteEn : REFERENCE TO BOOL;
	p_usiUSHermesReverseDSSendBFId : REFERENCE TO USINT;
	p_bUSHermesProcessRouteTrigger : REFERENCE TO BOOL;
	p_tySvyHermesSendWorkOrderInfo : REFERENCE TO tyHermesSendWorkOrderInfo;
	pa_RevtyXMLTableDataBrdAvl : REFERENCE TO ARRAY[0..200] OF tyXMLTableDat;
	p_ReviXMLTableDataBrdAvlTtlIdx : REFERENCE TO INT;
	p_bProcessRouteEn : REFERENCE TO BOOL;
	p_bReverseSentRoute : REFERENCE TO BOOL;
	p_bHermesSwitchtoRvrseTransport : REFERENCE TO BOOL;
END_VAR
(*Svy Hermes*)
VAR
	p_bManualInsertData : REFERENCE TO BOOL;
END_VAR
```

#### Local.var - Do Not Change!!!
```iecst
(*2020-09-10*)
(**)
(*Local Action, State & Status*)
VAR
	eAct : eHermesAction := HermesActIdle;
	eStat : eHermesAction := HermesActIdle;
	eMainStatus : eFBStatus := Idle;
	eStatus : eFBStatus := Idle;
	eStatus1 : eFBStatus := Idle;
	eStatus2 : eFBStatus := Idle;
	eStatus3 : eFBStatus := Idle;
	udiStatus : UDINT := 0;
	udiStatus1 : UDINT := 0;
	udiStatus2 : UDINT := 0;
	udiStatus3 : UDINT := 0;
	udiStatus4 : UDINT := 0;
	sStatTxt : STRING[200] := '';
	a_sStatText : ARRAY[0..50] OF STRING[200] := ['Idling','Background Starting Operations','Background Stopping Operations','Deleting Old Log File','Creating Directory','Writing Retain File','Reading Retain File','Saving Configuration',43('')];
END_VAR
(**)
(*Local Alarm*)
VAR
	tyAlmData : tyAlmDat;
	tyAlmData1 : tyAlmDat;
	tyAlmData2 : tyAlmDat;
	tyAlmData3 : tyAlmDat;
	tyAlmData4 : tyAlmDat;
	tyInfoData : tyAlmDat;
	a_tyAlmText : ARRAY[10000..10199] OF tyAlmTxt := [(sAlmText:='Invalid Ident While Creating Server',sRcyText:='Problem Occurred In The TCP/IP Connection. Check The Connection And Try To Reconnect.'),(sAlmText:='Setting Keep Alive Interval Time Error While Creating Server',sRcyText:='Unable To Establish Connection Between Machine. Check For Setting And Resume Operation.'),(sAlmText:='Setting Keep Alive Idle Time Error While Creating Server',sRcyText:='Unable To Establish Connection Between Machine. Check For Setting And Resume Operation.'),(sAlmText:='Setting Keep Alive Count Error While Creating Server',sRcyText:='Unable To Establish Connection Between Machine. Check For Setting And Resume Operation.'),(sAlmText:='Setting Keep Alive Error While Creating Server',sRcyText:='Unable To Establish Connection Between Machine. Check For Setting And Resume Operation.'),(sAlmText:='Setting Receive Buffer Error While Creating Server',sRcyText:='Unable To Establish Connection Between Machine. Check For Setting And Resume Operation.'),(sAlmText:='Setting Send Buffer Error While Creating Server',sRcyText:='Unable To Establish Connection Between Machine. Check For Setting And Resume Operation.'),(sAlmText:='Setting No Waiting Error While Creating Server',sRcyText:='Unable To Establish Connection Between Machine. Check For Setting And Resume Operation.'),(sAlmText:='TCP Open Port Error While Creating Server',sRcyText:='Problem Occurred In The TCP/IP Connection. Check The Connection And Try To Reconnect.'),(sAlmText:='Closing TCP Error While Creating Server',sRcyText:='Problem Occurred In The TCP/IP Connection. Check The Connection And Try To Reconnect.'),(sAlmText:='Invalid Ident While Listening Client',sRcyText:='There Was A Problem Connecting To The Server. The Server May Not Exist or It is Unavailable At This Time. Check The Connection and Try Again.'),(0),(sAlmText:='DS Hermes Connection Lost',sRcyText:='There Was A Problem Connecting To The Server. The Server May Not Exist or It is Unavailable At This Time. Check The Connection and Try Again.'),(0),(sAlmText:='Invalid Ident While Receiving Data',sRcyText:='Problem Occurred In The TCP/IP Connection. Check The Connection And Try To Reconnect.'),(sAlmText:='TCP Receive Data Error While Receiving Data',sRcyText:='Problem Occurred In The TCP/IP Connection. Check The Connection And Try To Reconnect.'),(sAlmText:='Receive BoardAvailable While Downstream In Not Connected State',sRcyText:='Receive Illegal Message.'),(sAlmText:='Receive RevokeBoardAvailable While Downstream In Not Connected State',sRcyText:='Receive Illegal Message.'),(sAlmText:='Receive MachineReady While Downstream In Not Connected State',sRcyText:='Receive Illegal Message.'),(sAlmText:='Receive RevokeMachineReady While Downstream In Not Connected State',sRcyText:='Receive Illegal Message.'),(sAlmText:='Receive StartTransport While Downstream In Not Connected State',sRcyText:='Receive Illegal Message.'),(sAlmText:='Receive StopTransport While Downstream In Not Connected State',sRcyText:='Receive Illegal Message.'),(sAlmText:='Receive TransportFinished While Downstream In Not Connected State',sRcyText:='Receive Illegal Message.'),(sAlmText:='Receive BoardForecast While Downstream In Not Connected State',sRcyText:='Receive Illegal Message.'),(sAlmText:='Receive ServiceDescription While Downstream In Service Description State',sRcyText:='Receive Illegal Message.'),(sAlmText:='Receive BoardAvailable While Downstream In Service Description State',sRcyText:='Receive Illegal Message.'),(sAlmText:='Receive RevokeBoardAvailable While Downstream In Service Description State',sRcyText:='Receive Illegal Message.'),(sAlmText:='Receive MachineReady While Downstream In Service Description State',sRcyText:='Receive Illegal Message.'),(sAlmText:='Receive RevokeMachineReady While Downstream In Service Description State',sRcyText:='Receive Illegal Message.'),(sAlmText:='Receive StartTransport While Downstream In Service Description State',sRcyText:='Receive Illegal Message.'),(sAlmText:='Receive StopTransport While Downstream In Service Description State',sRcyText:='Receive Illegal Message.'),(sAlmText:='Receive TransportFinished While Downstream In Service Description State',sRcyText:='Receive Illegal Message.'),(sAlmText:='Receive BoardForecast While Downstream In Service Description State',sRcyText:='Receive Illegal Message.'),(sAlmText:='Receive ServiceDescription While Downstream In Not Available Not Ready State',sRcyText:='Receive Illegal Message.'),(sAlmText:='Receive BoardAvailable While Downstream In Not Available Not Ready State',sRcyText:='Receive Illegal Message.'),(sAlmText:='Receive RevokeBoardAvailable While Downstream In Not Available Not Ready State',sRcyText:='Receive Illegal Message.'),(sAlmText:='Receive RevokeMachineReady While Downstream In Not Available Not Ready State',sRcyText:='Receive Illegal Message.'),(sAlmText:='Receive StartTransport While Downstream In Not Available Not Ready State',sRcyText:='Receive Illegal Message.'),(sAlmText:='Receive StopTransport While Downstream In Not Available Not Ready State',sRcyText:='Receive Illegal Message.'),(sAlmText:='Receive TransportFinished While Downstream In Not Available Not Ready State',sRcyText:='Receive Illegal Message.'),(sAlmText:='Receive BoardForecast While Downstream In Not Available Not Ready State',sRcyText:='Receive Illegal Message.'),(sAlmText:='Receive ServiceDescription While Downstream In Board Available State',sRcyText:='Receive Illegal Message.'),(sAlmText:='Receive BoardAvailable While Downstream In Board Available State',sRcyText:='Receive Illegal Message.'),(sAlmText:='Receive RevokeBoardAvailable While Downstream In Board Available State',sRcyText:='Receive Illegal Message.'),(sAlmText:='Receive RevokeMachineReady While Downstream In Board Available State',sRcyText:='Receive Illegal Message.'),(sAlmText:='Receive StartTransport While Downstream In Board Available State',sRcyText:='Receive Illegal Message.'),(sAlmText:='Receive StopTransport While Downstream In Board Available State',sRcyText:='Receive Illegal Message.'),(sAlmText:='Receive TransportFinished While Downstream In Board Available State',sRcyText:='Receive Illegal Message.'),(sAlmText:='Receive BoardForecast While Downstream In Board Available State',sRcyText:='Receive Illegal Message.'),(sAlmText:='Receive ServiceDescription While Downstream In Machine Ready State',sRcyText:='Receive Illegal Message.'),(sAlmText:='Receive BoardAvailable While Downstream In Machine Ready State',sRcyText:='Receive Illegal Message.'),(sAlmText:='Receive RevokeBoardAvailable While Downstream In Machine Ready State',sRcyText:='Receive Illegal Message.'),(sAlmText:='Receive MachineReady While Downstream In Machine Ready State',sRcyText:='Receive Illegal Message.'),(sAlmText:='Receive StopTransport While Downstream In Machine Ready State',sRcyText:='Receive Illegal Message.'),(sAlmText:='Receive TransportFinished While Downstream In Machine Ready State',sRcyText:='Receive Illegal Message.'),(sAlmText:='Receive BoardForecast While Downstream In Machine Ready State',sRcyText:='Receive Illegal Message.'),(sAlmText:='Receive ServiceDescription While Downstream In Available And Ready State',sRcyText:='Receive Illegal Message.'),(sAlmText:='Receive BoardAvailable While Downstream In Available And Ready State',sRcyText:='Receive Illegal Message.'),(sAlmText:='Receive RevokeBoardAvailable While Downstream In Available And Ready State',sRcyText:='Receive Illegal Message.'),(sAlmText:='Receive MachineReady While Downstream In Available And Ready State',sRcyText:='Receive Illegal Message.'),(sAlmText:='Receive StopTransport While Downstream In Available And Ready State',sRcyText:='Receive Illegal Message.'),(sAlmText:='Receive TransportFinished While Downstream In Available And Ready State',sRcyText:='Receive Illegal Message.'),(sAlmText:='Receive BoardForecast While Downstream In Available And Ready State',sRcyText:='Receive Illegal Message.'),(sAlmText:='Receive ServiceDescription While Downstream In Transporting State',sRcyText:='Receive Illegal Message.'),(sAlmText:='Receive BoardAvailable While Downstream In Transporting State',sRcyText:='Receive Illegal Message.'),(sAlmText:='Receive RevokeBoardAvailable While Downstream In Transporting State',sRcyText:='Receive Illegal Message.'),(sAlmText:='Receive MachineReady While Downstream In Transporting State',sRcyText:='Receive Illegal Message.'),(sAlmText:='Receive RevokeMachineReady While Downstream In Transporting State',sRcyText:='Receive Illegal Message.'),(sAlmText:='Receive StartTransport While Downstream In Transporting State',sRcyText:='Receive Illegal Message.'),(sAlmText:='Receive TransportFinished While Downstream In Transporting State',sRcyText:='Receive Illegal Message.'),(sAlmText:='Receive BoardForecast While Downstream In Transporting State',sRcyText:='Receive Illegal Message.'),(sAlmText:='Receive ServiceDescription While In Transport Finished State',sRcyText:='Receive Illegal Message.'),(sAlmText:='Receive BoardAvailable While In Transport Finished State',sRcyText:='Receive Illegal Message.'),(sAlmText:='Receive RevokeBoardAvailable While In Transport Finished State',sRcyText:='Receive Illegal Message.'),(sAlmText:='Receive MachineReady While In Transport Finished State',sRcyText:='Receive Illegal Message.'),(sAlmText:='Receive RevokeMachineReady While In Transport Finished State',sRcyText:='Receive Illegal Message.'),(sAlmText:='Receive StartTransport While In Transport Finished State',sRcyText:='Receive Illegal Message.'),(sAlmText:='Receive TransportFinished While In Transport Finished State',sRcyText:='Receive Illegal Message.'),(sAlmText:='Receive BoardForecast While In Transport Finished State',sRcyText:='Receive Illegal Message.'),(sAlmText:='Receive ServiceDescription While Downstream In Transport Stopped State',sRcyText:='Receive Illegal Message.'),(sAlmText:='Receive BoardAvailable While Downstream In Transport Stopped State',sRcyText:='Receive Illegal Message.'),(sAlmText:='Receive RevokeBoardAvailable While Downstream In Transport Stopped State',sRcyText:='Receive Illegal Message.'),(sAlmText:='Receive MachineReady While Downstream In Transport Stopped State',sRcyText:='Receive Illegal Message.'),(sAlmText:='Receive RevokeMachineReady While Downstream In Transport Stopped State',sRcyText:='Receive Illegal Message.'),(sAlmText:='Receive StartTransport While Downstream In Transport Stopped State',sRcyText:='Receive Illegal Message.'),(sAlmText:='Receive StopTransport While Downstream In Transport Stopped State',sRcyText:='Receive Illegal Message.'),(sAlmText:='LaneId Mismatch While Checking Service Description',sRcyText:='The LaneId Value Does Not Match. Change The Value And Resend The Value.'),(sAlmText:='MachineId Missing While Checking Service Description',sRcyText:='Missing Input Value For MachineId. Fill Up The Value And Resend.'),(sAlmText:='LandId Out Of Range While Checking Service Description',sRcyText:='LaneId Does Not Fall Within The Expected Range.'),(sAlmText:='LandId Missing While Checking Service Description',sRcyText:='Missing Input Value For LaneId. Fill Up The Value And Resend.'),(sAlmText:='Version Missing While Checking Service Description',sRcyText:='Missing Input Value For Version. Fill Up The Value And Resend.'),(sAlmText:='SupportedFeatures Missing While Checking Service Description',sRcyText:='Missing Input Value For SupportedFeatures. Fill Up The Value And Resend.'),(sAlmText:='NotificationCode Out Of Range While Checking Notification',sRcyText:='NotificationCode Does Not Fall Within The Expected Range.'),(sAlmText:='NotificationCode Missing While Checking Notification',sRcyText:='Missing Input Value For NotificationCode. Fill Up The Value And Resend.'),(sAlmText:='Severity Missing While Checking Notification',sRcyText:='Missing Input Value For Severity. Fill Up The Value And Resend.'),(sAlmText:='Description Missing While Checking Notification',sRcyText:='Missing Input Value For Description. Fill Up The Value And Resend.'),2((0)),(sAlmText:='FailedBoard Missing While Checking Machine Ready',sRcyText:='Missing Input Value For FailedBoard. Fill Up The Value And Resend.'),(sAlmText:='TransferState Missing While Checking Stop Transport',sRcyText:='Missing Input Value For TransferState. Fill Up The Value And Resend.'),(sAlmText:='BoardId Missing While Checking Stop Transport',sRcyText:='Missing Input Value For BoardId. Fill Up The Value And Resend.'),(sAlmText:='BoardId Missing While Checking Start Transport',sRcyText:='Missing Input Value For BoardId. Fill Up The Value And Resend.'),(sAlmText:='Barcode Missing While Checking Query Board Info',sRcyText:='Missing Input Value For BoardId. Fill Up The Value And Resend.'),(0),(sAlmText:='BoardId Mismatch While Checking Start Transport & Stop Transport',sRcyText:='The BoardId Value Does Not Match. Change The Value And Resend The Value.'),(sAlmText:='BoardId Missing While Checking Start Transport & Stop Transport',sRcyText:='Missing Input Value For BoardId. Fill Up The Value And Resend.'),(sAlmText:='Service Description Interchange Time Out',sRcyText:='Timeout Expired Before Operation Completed. Reset And Resume Operation.'),(sAlmText:='Transport Time Out',sRcyText:='Timeout Expired Before Operation Completed. Reset And Resume Operation.'),(sAlmText:='Receive TransportFinished While Downstream In Transport Stopped State',sRcyText:='Receive Illegal Message.'),(sAlmText:='Receive BoardForecast While Downstream In Transport Stopped State',sRcyText:='Receive Illegal Message.'),(sAlmText:='Stop Transport Request To Send From Upstream Hermes',sRcyText:='Sending Illegal Message.'),(sAlmText:='Get Directory Info Error While Deleting Old Log',sRcyText:='An Error Was Encountered While Getting Directory Info. Please Contact Nutek For A Possible Solution.'),(sAlmText:='Directory Read Error While Deleting Old Log',sRcyText:='An Error Was Encountered While Reading Directory. Please Contact Nutek For A Possible Solution.'),(sAlmText:='File Delete Error While Deleting Old Log',sRcyText:='An Error Was Encountered While Trying To Delete File. Please Contact Nutek For A Possible Solution.'),18((0)),(sAlmText:='Check Alive Time Out',sRcyText:='Timeout Expired Before Operation Completed. Reset And Resume Operation.'),(sAlmText:='Waiting Check Alive Time Out',sRcyText:='Timeout Expired Before Operation Completed. Reset And Resume Operation.'),(sAlmText:='Check Alive Id Mismatch',sRcyText:='The Check Alive Id Value Does Not Match. Change The Value And Resend The Value.'),(sAlmText:='Machine Ready Request To Send From Upstream Hermes',sRcyText:='Sending Illegal Message.'),(sAlmText:='Revoke Machine Ready Request To Send From Upstream Hermes',sRcyText:='Sending Illegal Message.'),(sAlmText:='Start Transport Request To Send From Upstream Hermes',sRcyText:='Sending Illegal Message.'),(sAlmText:='Set Configuration Request To Send From Upstream Hermes',sRcyText:='Sending Illegal Message.'),(sAlmText:='Get Configuration Request To Send From Upstream Hermes',sRcyText:='Sending Illegal Message.'),(sAlmText:='Current Configuration Request To Send From Upstream Hermes',sRcyText:='Sending Illegal Message.'),(sAlmText:='Board Forecast Request To Send From Upstream Hermes',sRcyText:='Sending Illegal Message.'),(sAlmText:='Query Board Info Request To Send From Upstream Hermes',sRcyText:='Sending Illegal Message.'),(sAlmText:='Invalid Ident While Sending Data',sRcyText:='Invalid Ident Value.'),(sAlmText:='TCP Retry Send Data Error While Sending Data',sRcyText:='Problem Occurred In The TCP/IP Connection. Check The Connection And Try To Reconnect.'),(sAlmText:='TCP Send Data Error',sRcyText:='Problem Occurred In The TCP/IP Connection. Check The Connection And Try To Reconnect.'),(sAlmText:='Invalid Ident While Closing TCP',sRcyText:='Invalid Ident Value.'),(sAlmText:='Closing TCP Error',sRcyText:='Problem Occurred In The TCP/IP Connection. Check The Connection And Try To Reconnect.'),(sAlmText:='File Open Error While Writing Log',sRcyText:='An Error Was Encountered While Trying To Open File. Please Contact Nutek For A Possible Solution.'),(sAlmText:='File Create Error While Writing Log',sRcyText:='An Error Was Encountered While Trying To Create File. Please Contact Nutek For A Possible Solution.'),(sAlmText:='Get File Info Error While Writing Log',sRcyText:='An Error Was Encountered While Getting File Info. Please Contact Nutek For A Possible Solution.'),(sAlmText:='File Write Error While Writing Log',sRcyText:='An Error Was Encountered While Trying To Write File. Please Contact Nutek For A Possible Solution.'),(sAlmText:='File Close Error While Writing Log',sRcyText:='An Error Was Encountered While Trying To Close File. Please Contact Nutek For A Possible Solution.'),(sAlmText:='Directory Does Not Exist While Writing Log',sRcyText:='The Directory Does Not Exist.Please Contact Nutek For A Possible Solution.'),(sAlmText:='Invalid Ident While Closing TCP',sRcyText:='Invalid Ident Value.'),(sAlmText:='Closing TCP Error',sRcyText:='Problem Occurred In The TCP/IP Connection. Check The Connection And Try To Reconnect.'),(0),(sAlmText:='Board Jam At Sensor After Transfer Interrupted',sRcyText:='Pull Back Board From Downstream Machine'),42((0))];
END_VAR
(**)
(*Local Output*)
VAR
	bConnected : BOOL;
	bHandshakeDone : BOOL;
	bUSRdy : BOOL;
	bDSRdy : BOOL;
	bUSGdRdy : BOOL;
	bDSGdRdy : BOOL;
	bTransporting : BOOL;
	bStopTransport : BOOL;
	sInternalSnd : STRING[65535];
END_VAR
(**)
(*Local Input*)
VAR
	udiRstErr : UDINT := 0;
	bPrep : BOOL := TRUE;
	bEn : BOOL := TRUE;
	bDis : BOOL := FALSE;
	tyParam : tyHermesDSParam;
	sIPAddr : STRING[15] := '192.168.0.100';
	a_usiMacAddr : ARRAY[0..5] OF USINT := [6(0)];
	tyDTStructure : DTStructure := (year:=2019,month:=01,day:=05,wday:=05,hour:=21,minute:=28,second:=30,millisec:=123,microsec:=456);
	dtCurrDT : DATE_AND_TIME := DT#2019-02-23-12:30:50;
	bRdySnd : BOOL := FALSE;
	bSndCompl : BOOL := FALSE;
	bSndInCompl : BOOL := FALSE;
	bSndNotStart : BOOL := FALSE;
	bBAWidthEn : BOOL := TRUE; (*Board Available Check Width*)
	bBASltEn : BOOL := FALSE; (*Board Available Check Slot*)
	bBFWidthEn : BOOL := TRUE; (*Board Available Check Width*)
	bBFSltEn : BOOL := FALSE; (*Board Available Check Slot*)
	sMcId : STRING[80] := '';
	sInterfaceId : STRING[80];
	sVersion : STRING[7] := '1.0.2';
	eFailedBoard : eHermesFailedBoard := HermesUnknownBoard;
	sRecipeNm : STRING[254] := '';
	eFlippedBoard : eHermesFlippedBoard := HermesFlippedBoardUnknownSide;
	sTopBarcode : STRING[254] := '';
	sBottomBarcode : STRING[254] := '';
	rLength : REAL := 0;
	rThickness : REAL := 0;
	rConveyorSpeed : REAL := 0;
	rTopClearanceHeight : REAL := 0;
	rBottomClearanceHeight : REAL := 0;
	rWeight : REAL := 0;
	sWorkOrderId : STRING[80] := '';
	sBatchId : STRING[80] := '';
	diWidthInUM : DINT := 0;
	diMinSltValue : DINT := 0;
	diMaxSltValue : DINT := 0;
	diPitch : DINT := 0;
	diTtlSlt : DINT := 0;
	diSltToSltInUM : DINT := 0;
	udiSndBffrSize : UDINT := 65536;
	udiRcvBffrSize : UDINT := 65536;
	udiAliveIdleTimeInSec : UDINT := 5;
	tConnTimeOut : TIME := T#30s;
	diTransferInTO : DINT := 30000;
	a_tyXMLTableDataBrdAvl : ARRAY[0..200] OF tyXMLTableDat;
	iXMLTableDataBrdAvlTtlIdx : INT := 0;
	bNewBrdAvl : BOOL := FALSE;
	bOpsRun : BOOL := FALSE;
	bInterruptSen : BOOL := FALSE;
	udiFileKeepDay : UDINT := 30;
	sProgNm : STRING[15] := 'DSHermes';
	bNtSettingsLoadDone : BOOL := TRUE;
	sRmtMcId : STRING[80];
	bRmtPrep : BOOL := FALSE;
	bRmtEn : BOOL := FALSE;
	bInternalUse : BOOL;
	sInternalRcv : STRING[65535];
END_VAR
(**)
(*Local*)
VAR
	bRstErr : BOOL;
	udiRstErrOld : UDINT;
	bInitDone : BOOL;
	bInitialDone : BOOL;
	bRun : BOOL;
	bStop : BOOL;
	bRstConnection : BOOL;
	bRstState : BOOL;
	udiSvrIdent : UDINT;
	udiClntIdent : UDINT;
	udiClntIdentExtra : UDINT;
	udiXMLTableWriteIdx : UDINT;
	udiMsgSendBffr : UDINT;
	udiMsgCmdBffr : UDINT;
	udiSndMsgLen : UDINT;
	sSnd : STRING[65535];
	sRcv : STRING[65535];
	a_tyXMLTableDataRcv : ARRAY[0..200] OF tyXMLTableDat;
	a_tyXMLTableDataSnd : ARRAY[0..200] OF tyXMLTableDat;
	a_eMsgSend : ARRAY[0..50] OF eHermesMsgType;
	a_eCommandSndQ : ARRAY[0..20] OF eHermesCommand;
	tyMsgTypeRcv : tyHermesMsgType;
	tyCheckAliveSnd : tyHermesCheckAlive;
	tyCheckAlivePingSnd : tyHermesCheckAlive;
	tyCheckAlivePongSnd : tyHermesCheckAlive;
	tyCheckAliveRcv : tyHermesCheckAlive;
	tyCheckAlivePingRcv : tyHermesCheckAlive;
	tyCheckAlivePongRcv : tyHermesCheckAlive;
	tyServiceDescriptionSnd : tyHermesServiceDescription;
	tyServiceDescriptionRcv : tyHermesServiceDescription;
	tyNotificationSnd : tyHermesNotification;
	tyNotificationRcv : tyHermesNotification;
	tyBoardAvailableRcv : tyHermesBoardAvailable;
	tyBoardAvailableSnd : tyHermesBoardAvailable;
	a_tyBoardDepartedInfo : ARRAY[0..49] OF tyHermesBoardAvailable;
	a_tyBoardDepartedInfoWr : ARRAY[0..49] OF tyHermesBoardAvailable;
	tyMachineReady : tyHermesMachineReady;
	tyStartTransport : tyHermesStartTransport;
	tyStopTransport : tyHermesStopTransport;
	tyTransportFinished : tyHermesTransportFinished;
	tySetConfiguration : tyHermesSetConfiguration;
	tyCurrentConfiguration : tyHermesCurrentConfiguration;
	tyBoardForecastRcv : tyHermesBoardForecast;
	tyBoardForecastSnd : tyHermesBoardForecast;
	tyQueryBoardInfo : tyHermesQueryBoardInfo;
	tySendBoardInfo : tyHermesSendBoardInfo;
	tyCommandRcv : tyHermesCommand;
	tyCommandSnd : tyHermesCommand;
	fbCreateSvr : fbTCPCreateSvr;
	fbListen : fbTCPListen;
	fbRcv : fbTCPRcv;
	fbSend : fbTCPSnd;
	fbCloseSvr : fbTCPClose;
	fbCloseClnt : fbTCPClose;
	fbParseXMLTable : fbHermesParseXMLTable;
	fbParseBrdAvlExternal : fbHermesParseXMLTable;
	fbCheckAlive : fbHermesCheckAlive;
	fbCheckAliveSendPing : fbHermesCheckAliveSendPing;
	fbCheckAliveRcvPing : fbHermesCheckAliveRcvPing;
	fbSequenceDS : fbHermesSequenceDS;
	fbSequenceTO : fbHermesSequenceTO;
END_VAR
VAR RETAIN
	usiBAIndex : USINT := 0;
END_VAR
VAR
	usiPrevBAIndex : USINT;
	eStatOld : eHermesAction := HermesActIdle;
	tyParamOld : tyHermesDSParam;
	udiLogCntr : UDINT := 1;
	udiWriteLogCntr : UDINT := 1;
	a_sLogList : ARRAY[1..10] OF STRING[65535];
	sDT : STRING[80];
	dtCurrDTTemp : DATE_AND_TIME;
	fbFileAppend1 : fbFileFullAppend;
	fbFileOldDel1 : fbFileOldDel;
	fbFileRead1 : fbFileFullRead;
	fbFileWrite1 : fbFileFullWrite;
	iWriteLogStep : INT := 0;
	tyUSHermestyBoardAvailable : tyHermesBoardAvailable;
	tyCommandParam : tyHermesCommandParam;
	bDummy : BOOL;
	bFeatureBoardForecast : BOOL;
	bNewProduct : BOOL;
	bNewWidth : BOOL;
	bNewChangeOver : BOOL;
	tySendBoardInfoAcc : tyHermesSendBoardInfo;
	rMachineCycleTime : REAL;
	rAWCycleTm : REAL;
	bFileNotFound : BOOL;
	bSendBFId : BOOL;
	bBFIdSent : BOOL;
	bSendBFNoID : BOOL;
	bSndReverseBF : BOOL;
	bRstSendBFId : BOOL;
	bFirstZoneHaveBoard : BOOL;
	bFirstZoneEndSen : BOOL;
	bAllZoneEmpty : BOOL;
	bTransportFinishedSnd : BOOL;
	fbTimerRstBFId : TON;
	sInfoMcRdyMsg : STRING[200];
	sTempRealWidth : STRING[15];
	sRstTim : STRING[15];
	udiModuleNum : UDINT := 3351;
END_VAR
(*Send Board Info*)
VAR
	bSearchTop : BOOL;
	bSearchBottom : BOOL;
	siTopBarcodeIdx : SINT;
	siBottomBarcodeIdx : SINT;
	siSearhIdx : SINT;
	siFoundIdx : SINT;
	bCompleteSearch : BOOL;
END_VAR
(*Route*)
VAR
	bTriggerRouteReversal : BOOL;
	bReverseDSSndBfWBrdID : BOOL;
	bSwitchtoReverseSend : BOOL;
	fbRstReverseSndGate : TON;
	bNotifyRstReverseSndGate : BOOL;
	bBlkDS : BOOL;
	bProcessRouteEn : BOOL;
	bManualRmvRoute : BOOL;
	bReturnRoute : BOOL;
	bNomRouteEn : BOOL;
	bReverseSentRoute : BOOL;
	usiUSHermesReverseDSSendBFId : USINT;
	bUSHermesProcessRouteTrigger : BOOL;
	iRoute : INT;
	iAction : INT;
	bDSHermesRcvReverseUSMcRdy : BOOL;
	bReverseRcvBlkDS : BOOL;
	bTest1 : BOOL;
	bTest2 : BOOL;
END_VAR
```

### DSHermes2.var - Change By Project
```iecst
(*2020-09-10*)
(**)
(*Action & State & Status*)
VAR
	p_DSHermes2Stat : UDINT;
	p_DSHermes2Status : UDINT;
	p_DSHermes2StatTxt : UDINT;
END_VAR
(**)
(*Alarm*)
VAR
	p_DSHermes2AlmData : UDINT;
	p_DSHermes2AlmData1 : UDINT;
	p_DSHermes2AlmData2 : UDINT;
	p_DSHermes2AlmData3 : UDINT;
	p_DSHermes2AlmData4 : UDINT;
END_VAR
(**)
(*Output*)
VAR
	p_DSHermes2Connected : UDINT;
	p_DSHermes2HandshakeDone : UDINT;
	p_DSHermes2USRdy : UDINT;
	p_DSHermes2DSRdy : UDINT;
	p_DSHermes2USGdRdy : UDINT;
	p_DSHermes2DSGdRdy : UDINT;
	p_DSHermes2Transporting : UDINT;
	p_DSHermes2StopTransport : UDINT;
	p_DSHermes2InternalSnd : UDINT;
	p_DSHermes2CommandParam : UDINT;
	p_DSHermes2BrdAvlSnd : UDINT;
	p_DSHermes2TransportFinish : UDINT;
	p_DSHermes2TransportFinishMsg : UDINT;
END_VAR
```

### Program Logical/Hermes/DSHermes2 (IEC) - 1.00.0 - NtHermes v5.00.0 , NtTCP v5.00.0 , NtMessage v5.00.0

#### InputRef.var
```iecst
(*2019-06-10*)
(**)
(*General*)
VAR
	p_eAct : REFERENCE TO eHermesAction;
	p_udiRstErr : REFERENCE TO UDINT;
	p_bPrep : REFERENCE TO BOOL;
	p_bEn : REFERENCE TO BOOL;
	p_bDis : REFERENCE TO BOOL;
END_VAR
(**)
(*Configuration*)
VAR
	p_tyParam : REFERENCE TO tyHermesDSParam;
	p_sIPAddr : REFERENCE TO STRING[15];
	pa_usiMacAddr : REFERENCE TO ARRAY[0..5] OF USINT;
	p_tyDTStructure : REFERENCE TO DTStructure;
	p_dtCurrDT : REFERENCE TO DATE_AND_TIME;
	p_sMcId : REFERENCE TO STRING[80];
END_VAR
(**)
(*Input*)
VAR
	p_bRdySnd : REFERENCE TO BOOL;
	p_bSndCompl : REFERENCE TO BOOL;
	p_bSndIncompl : REFERENCE TO BOOL;
	p_bSndNotStart : REFERENCE TO BOOL;
	p_bBAWidthEn : REFERENCE TO BOOL; (*Board Available Check Width*)
	p_bBASltEn : REFERENCE TO BOOL; (*Board Available Check Slot*)
	p_bBFWidthEn : REFERENCE TO BOOL; (*Board Forecast Check Width*)
	p_bBFSltEn : REFERENCE TO BOOL; (*Board Forecast Check Slot*)
	p_sRecipeNm : REFERENCE TO STRING[254];
	p_sRecipeZone1Nm : REFERENCE TO STRING[254];
	p_sForecastId : REFERENCE TO STRING[80];
	p_sBoardId : REFERENCE TO STRING[36];
	p_sInterfaceId : REFERENCE TO STRING[80];
	p_sVersion : REFERENCE TO STRING[7];
	p_eFailedBoard : REFERENCE TO eHermesFailedBoard;
	p_eFlippedBoard : REFERENCE TO eHermesFlippedBoard;
	p_sTopBarcode : REFERENCE TO STRING[254];
	p_sBottomBarcode : REFERENCE TO STRING[254];
	p_rLength : REFERENCE TO REAL;
	p_rThickness : REFERENCE TO REAL;
	p_rConveyorSpeed : REFERENCE TO REAL;
	p_rTopClearanceHeight : REFERENCE TO REAL;
	p_rBottomClearanceHeight : REFERENCE TO REAL;
	p_rWeight : REFERENCE TO REAL;
	p_sWorkOrderId : REFERENCE TO STRING[80];
	p_sBatchId : REFERENCE TO STRING[80];
	p_diWidthInUM : REFERENCE TO DINT;
	p_diWidthZone1InUM : REFERENCE TO DINT;
	p_diMinSltValue : REFERENCE TO DINT;
	p_diMaxSltValue : REFERENCE TO DINT;
	p_diPitch : REFERENCE TO DINT;
	p_diTtlSlt : REFERENCE TO DINT;
	p_diSltToSltInUM : REFERENCE TO DINT;
	p_udiSndBffrSize : REFERENCE TO UDINT;
	p_udiRcvBffrSize : REFERENCE TO UDINT;
	p_udiAliveIdleTimeInSec : REFERENCE TO UDINT;
	p_tConnTimeOut : REFERENCE TO TIME;
	p_diTransferInTO : REFERENCE TO DINT;
	pa_tyXMLTableDataBrdAvl : REFERENCE TO ARRAY[0..200] OF tyXMLTableDat;
	p_iXMLTableDataBrdAvlTtlIdx : REFERENCE TO INT;
	p_bNewBrdAvlFirstZone : REFERENCE TO BOOL;
	p_bNewBrdAvlLastZone : REFERENCE TO BOOL;
	p_bOpsRun : REFERENCE TO BOOL;
	p_bInterruptSen : REFERENCE TO BOOL;
	p_udiFileKeepDay : REFERENCE TO UDINT;
	p_udiRetainDataAddr : REFERENCE TO UDINT;
	p_udiRetainDataLen : REFERENCE TO UDINT;
	p_sRetainFileName : REFERENCE TO STRING[80];
	p_sProgNm : REFERENCE TO STRING[15];
	p_bNtSettingsLoadDone : REFERENCE TO BOOL;
	p_sRmtMcId : REFERENCE TO STRING[80];
	p_bRmtPrep : REFERENCE TO BOOL;
	p_bRmtEn : REFERENCE TO BOOL;
	p_bUSHermesStopTransport : REFERENCE TO BOOL;
	p_bInternalUse : REFERENCE TO BOOL;
	p_sInternalRcv : REFERENCE TO STRING[65535];
	p_tyUSBoardArrivedData : REFERENCE TO tyHermesBoardAvailable;
	p_bRcvBoardInfo : REFERENCE TO BOOL;
	p_tyBoardInfoData : REFERENCE TO tyHermesSendBoardInfo;
	p_tyUSHermestyBoardAvailable : REFERENCE TO tyHermesBoardAvailable;
	p_bNtParamProjInvertOncePrep : REFERENCE TO BOOL;
	p_bNtParamProjInvertTwicePrep : REFERENCE TO BOOL;
	p_bReverseDSSendBFId : REFERENCE TO BOOL;
	p_rMcCycleTm : REFERENCE TO REAL;
	p_rAWCycleTm : REFERENCE TO REAL;
	p_bConvInitDone : REFERENCE TO BOOL;
END_VAR
(*Reverse Hermes *)
VAR
	p_bManualRmvRoute : REFERENCE TO BOOL;
	p_bReturnRoute : REFERENCE TO BOOL;
	p_bNomRouteEn : REFERENCE TO BOOL;
	p_usiUSHermesReverseDSSendBFId : REFERENCE TO USINT;
	p_bUSHermesProcessRouteTrigger : REFERENCE TO BOOL;
	p_tySvyHermesSendWorkOrderInfo : REFERENCE TO tyHermesSendWorkOrderInfo;
	pa_RevtyXMLTableDataBrdAvl : REFERENCE TO ARRAY[0..200] OF tyXMLTableDat;
	p_ReviXMLTableDataBrdAvlTtlIdx : REFERENCE TO INT;
	p_bProcessRouteEn : REFERENCE TO BOOL;
	p_bReverseSentRoute : REFERENCE TO BOOL;
	p_bHermesSwitchtoRvrseTransport : REFERENCE TO BOOL;
END_VAR
(*Svy Hermes*)
VAR
	p_bManualInsertData : REFERENCE TO BOOL;
END_VAR
```
